FUNCTION F_CoolTank 
VAR_INPUT
	rTank : REFERENCE TO ST_Tank;
END_VAR
VAR
	
END_VAR

IF __ISVALIDREF(rTank) THEN
	IF rTank.fTemperature > GVL.GC_TARGET_TEMPERATURE THEN
		rTank.fTemperature := rTank.fTemperature - GVL.GC_COOLING_RATE;
	ELSE
		rTank.bTemperatureAlarm := FALSE;
	END_IF
END_IF

END_FUNCTION

(* stored: Version 1.1.0.1, ProductVersion 3.1.4024.16
   POU F_CoolTank: Id {1f0e7e1c-76a6-4d5d-b4ea-ed11eac8e562}, SpecialFunc None *)
